VAR_GLOBAL
    astAxes				: 	ARRAY [1..GVL_APP.nAXIS_NUM] OF ST_AxisStruct; //Global array of ST_AxisStruct for holding axis parameters and controls
    iAxis				: 	UINT; //Index for for loops while going through axes
END_VAR

VAR_GLOBAL CONSTANT
    nMAX_AXIS_NAME		: 	UINT := 32;
END_VAR

VAR_GLOBAL PERSISTENT
    astAxesPersistent	: 	ARRAY [1..GVL_APP.nAXIS_NUM] OF ST_AxisPersistent;
END_VAR

(* stored: Version 1.1.0.1, ProductVersion 3.1.4024.5
   GVL GVL: Id {913e21aa-a47e-444c-bfce-679b16c0434b} *)
